TYPE OutputBase_10CEE7DE :
STRUCT
END_STRUCT
END_TYPE

(* stored: Version 1.2.0.0, ProductVersion 3.1.4024.11
   DUT OutputBase_10CEE7DE: Id {d591baf1-f8c5-4f4e-bb02-a2d4e04cf0b6} *)
